// TIA Portal V21 export
TYPE "LAxisCtrl_typeHaltSuperimposed"
TITLE = LAxisCtrl_typeHaltSuperimposed
// Support: tech.team.motioncontrol@siemens.com
   STRUCT
      deceleration : LReal := -1.0;   // Deceleration of the superimposed motion (Value > 0.0: The specified value is used; Value = 0.0: Not permitted; Value < 0.0: The deceleration configured in "Technology object > Configuration > Extended parameters > Dynamic default values" is used. <TO>.DynamicDefaults.Deceleration)
      jerk : LReal := -1.0;   // Jerk of the superimposed motion (Value > 0.0: Constant-acceleration velocity profile of the superimposed motion; the specified jerk is used; Value = 0.0: Trapezoidal velocity profile of the superimposed motion; Value < 0.0: The jerk configured in "Technology object > Configuration > Extended parameters > Dynamic default values" is used. <TO>.DynamicDefaults.Jerk)
      abortAcceleration : Bool := FALSE;   // TRUE: The acceleration of the superimposed motion is set to 0.0 at the start of the job, the deceleration builds up immediately; FALSE: The current acceleration of the superimposed motion at the start of the job is reduced using the configured jerk. Afterwards, the deceleration builds up
   END_STRUCT;
END_TYPE
